{attribute 'no_explicit_call':= 'do not call this POU directly'}
FUNCTION_BLOCK TValueMonitor
VAR
    _CurrentValue : INT := -1;
    _PreviousValue : INT;
    _Changed : BOOL;
END_VAR

PROPERTY Changed : BOOL
GET
Changed := _Changed;
END_GET
END_PROPERTY

PROPERTY CurrentValue : INT
GET
CurrentValue := _CurrentValue;
END_GET
END_PROPERTY

PROPERTY PreviousValue : INT
GET
PreviousValue := _PreviousValue;
END_GET
END_PROPERTY

METHOD Reset
VAR_INPUT
END_VAR
_CurrentValue := 0;
_PreviousValue := 0;
END_METHOD

METHOD Test : BOOL
VAR_INPUT
    Value : INT;
END_VAR
_Changed := Value <> _CurrentValue;
_PreviousValue := _CurrentValue;
_CurrentValue := Value;

Test := _Changed;
END_METHOD

END_FUNCTION_BLOCK

(* stored: Version 1.1.0.1, ProductVersion 3.1.4024.3
   POU TValueMonitor: Id {3e30235b-556e-0cbb-38fe-867062101222}, SpecialFunc None
   Property Changed: Id {6e0eabef-a51f-0aa9-227c-35902feaa60a}
   Get Get: Id {bee77674-8a70-054e-0110-6b95c1045f45}
   Property CurrentValue: Id {1060c0f1-95b1-010b-3cf3-d67b1d10a3f2}
   Get Get: Id {4f95a500-9447-09af-1099-7b8b5a55f72a}
   Property PreviousValue: Id {a339600b-a845-0a1d-2f9b-029c78ee027f}
   Get Get: Id {d3d603e7-26f5-07a2-2d51-d96700ba8064}
   Method Reset: Id {f34d3a68-4510-0aca-1fbc-e57e2410f56f}
   Method Test: Id {6529cf7b-ec45-0f00-18ca-636102b11808} *)
